Staubli VAL3: CSHAPE.pgx

public program Cshape(trsf& x_Source[], trsf& x_trCut[], num x_nAngle, num& x_nPointCout, trsf x_trCen, num x_nDia, bool& x_bRes)
  local trsf l_trTrsf[3]
  local num l_nNum
  local num l_nBuff
  local trsf l_trBuff
  local frame l_fFrame
begin

  //C型图形
  x_bRes=false
  if x_nAngle<=0 or x_nAngle>3600

    return
  endIf

  //由于TRSF.RZ的范围是 +-360


  l_trTrsf[0]=x_trCen
  l_trTrsf[1]=x_Source[0]
  l_trTrsf[2]=x_Source[1]

  // x_trCut[0]=x_Source[0]
  call SetFrame(l_trTrsf,l_fFrame,x_bRes)
  if !x_bRes
    return
  endIf


  x_nPointCout=roundUp(x_nAngle/180)+1
  x_nDia=x_nDia/2
  l_nBuff=x_nAngle/(x_nPointCout-1)/2
//  nNum=l_nBuff
  x_trCut[0]=l_fFrame.trsf*{x_nDia,0,0,0,0,0}
  for l_nNum=0 to x_nPointCout-2
    x_trCut[l_nNum*2+1]=l_fFrame.trsf*{cos((l_nNum*2+1)*l_nBuff)*x_nDia,sin((l_nNum*2+1)*l_nBuff)*x_nDia,0,0,0,0}
    x_trCut[l_nNum*2+2]=l_fFrame.trsf*{cos((l_nNum*2+2)*l_nBuff)*x_nDia,sin((l_nNum*2+2)*l_nBuff)*x_nDia,0,0,0,0}

  endFor


  x_bRes=true




end
